// TIA Portal V15.1 export
// export: Created 2024-06-21T08:40:52.7405115Z, ExportSetting WithDefaults, DisplayName Totally Integrated Automation Portal, DisplayVersion V15.1 Update 5, DisplayName TIA Portal Openness, DisplayVersion V15.1 Update 5, DisplayName SINAMICS Startdrive Advanced, DisplayVersion V15.1, DisplayName G130, G150, S120, S150, SINAMICS MV, S210, DisplayVersion V15.1, DisplayName G110M, G120, G120C, G120D, G120P, DisplayVersion V15.1, DisplayName STEP 7 Professional, DisplayVersion V15.1 Update 5, DisplayName STEP 7 Safety, DisplayVersion V15.1, DisplayName WinCC Professional, DisplayVersion V15.1 Update 5, DisplayName SIMATIC Visualization Architect, DisplayVersion V15.1
FUNCTION_BLOCK "LToggle"   // FB1108, FBD
TITLE = LToggle
{ S7_Optimized_Access := 'TRUE' }
AUTHOR : VCC
FAMILY : Function
NAME : LToggle
VERSION : 0.1
// ================================================================================
// Change the state of the output everytime the input is on
// ================================================================================
// stored: AutoNumber false, IsIECCheckEnabled false, IsRetainMemResEnabled false, MemoryReserve 100, SetENOAutomatically False, UDAEnableTagReadback false
   VAR_INPUT
      I_Input { ExternalAccessible := 'False'; ExternalVisible := 'False'; ExternalWritable := 'False'} : Bool;   // The input
   END_VAR
   VAR_OUTPUT
      O_Output { ExternalAccessible := 'False'; ExternalVisible := 'False'; ExternalWritable := 'False'} : Bool;   // The output
   END_VAR
   VAR RETAIN
      pulseReqOn { ExternalAccessible := 'False'; ExternalVisible := 'False'; ExternalWritable := 'False'} : Bool;   // Pulse request on
      pulseReqOff { ExternalAccessible := 'False'; ExternalVisible := 'False'; ExternalWritable := 'False'} : Bool;   // Pulse request off
      Output { ExternalAccessible := 'False'; ExternalVisible := 'False'; ExternalWritable := 'False'} : Bool;   // Temporary Output
      ReqOutputOff { ExternalAccessible := 'False'; ExternalVisible := 'False'; ExternalWritable := 'False'} : Bool;   // Request output off
      ReqOutputOn { ExternalAccessible := 'False'; ExternalVisible := 'False'; ExternalWritable := 'False'} : Bool;   // Request output on
   END_VAR
   VAR_TEMP   // added for the SCL form of the ladder/FBD networks
      _w1 : Bool;
   END_VAR
BEGIN

REGION Network 1: **** 5.2 - Equations - Flow **** Request on
   // Request on
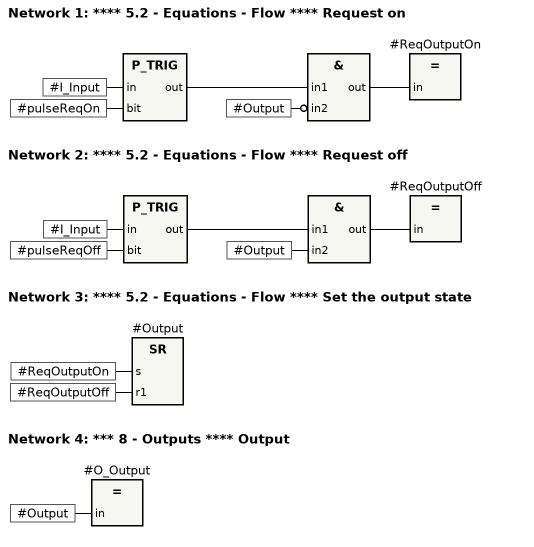
   #_w1 := #I_Input AND NOT #pulseReqOn;   // rising edge
   #pulseReqOn := #I_Input;
   #ReqOutputOn := #_w1 AND NOT #Output;
END_REGION

REGION Network 2: **** 5.2 - Equations - Flow **** Request off
   // Request off
   #_w1 := #I_Input AND NOT #pulseReqOff;   // rising edge
   #pulseReqOff := #I_Input;
   #ReqOutputOff := #_w1 AND #Output;
END_REGION

REGION Network 3: **** 5.2 - Equations - Flow **** Set the output state
   // Set the output state
   IF #ReqOutputOn THEN
       #Output := TRUE;   // SR flip-flop
   END_IF;
   IF #ReqOutputOff THEN #Output := FALSE; END_IF;
END_REGION

REGION Network 4: *** 8 - Outputs **** Output
   // Output
   #O_Output := #Output;
END_REGION
END_FUNCTION_BLOCK
